FUNCTION_BLOCK FB_BagOpener
VAR_INPUT
  ams_net_id	: STRING;
END_VAR
VAR_OUTPUT
END_VAR
VAR
	adsread				: ADSREAD;
	adswrite			: ADSWRITE;
	status				: BagMachineStatus;
	iMethodTest			: BagMachineStatus;
	bagOpenStatus 		: BagMachineStatus;
  	error_code			: UINT;

	adsArr				: AdsArr;
	iState				: INT;
	iAds				: INT;
	ton_ms				: TON;
	iMachineStatus		: INT;//inArr[0]
	iBagStatus			: INT;//inArr[1]
	iBagDetectStatus	: INT;//inArr[2]
	iBagCmd				: INT;//outArr[1]
	iBagDetectCmd		: INT;//outArr[2]
	
	
	
END_VAR

	adsread(
			NETID:=ams_net_id , 
			PORT:=851 , 
			IDXGRP:=16#00004020 , 
			IDXOFFS:=100 , 
			LEN:= SIZEOF(adsArr.inArr), 
			DESTADDR:= ADR(adsArr.inArr), 
			READ:=, 
			TMOUT:=T#2S , 
			BUSY=> , 
			ERR=> , 
			ERRID=> );
	adswrite(
			NETID:=ams_net_id , 
			PORT:=851, 
			IDXGRP:=16#00004020, 
			IDXOFFS:=200, 
			LEN:=SIZEOF(adsArr.outArr) , 
			SRCADDR:=ADR(adsArr.outArr) , 
			WRITE:= , 
			TMOUT:=T#2S , 
			BUSY=> , 
			ERR=> , 
			ERRID=> );
ton_ms(PT:=T#2MS);			
CASE iAds OF 
	0:
		adsread.READ	:= FALSE;
		adswrite.WRITE	:= FALSE;	
		iAds	:=1;
	1:
		ton_ms.IN	:= TRUE;
		IF ton_ms.Q THEN
			ton_ms.IN	:= FALSE;
			iAds	:=2;
		END_IF
	2:
		adsread.READ	:= TRUE;
		adswrite.WRITE	:= TRUE;
		iAds	:=3;
	3:
		ton_ms.IN	:= TRUE;
		IF ton_ms.Q THEN
			ton_ms.IN	:= FALSE;
			iAds	:=0;
		END_IF	
END_CASE
//inputArr:
//		[0]:machine status;
//		[1]:bag status(3:BAG_READY,4:BAG_INSERTED,5:BAG_REMOVED,6:camera_ok,7:camera_ng);
//		[2]:bag detect status(0:idle,1:ok,2:ng);	
//outputArr:
//		[0]:line status;
//		[1]:bag cmd(1:insert_bag,2:bag_done_clamping,3:camera_trigger,4:camera_reset);
//	    [2]:bag detect cmd(0:idle,1:trigger,2:reset);
iMachineStatus		:= WORD_TO_INT(adsArr.inArr[0]);
iBagStatus 			:= WORD_TO_INT(adsArr.inArr[1]);
iBagDetectStatus	:= WORD_TO_INT(adsArr.inArr[2]);
adsArr.outArr[1]	:= INT_TO_WORD(iBagCmd);
adsArr.outArr[2]	:= INT_TO_WORD(iBagDetectCmd);

CASE iMachineStatus OF
	0:
		status	:= BagMachineStatus.OFF;
	1:
		status	:= BagMachineStatus.READY;
	2:
		status	:= BagMachineStatus.BUSY;
	3:
		status	:= BagMachineStatus.ERROR;
END_CASE
CASE iMethodTest OF
	BagMachineStatus.OFF:
		iState	:= BagMachineStatus.OFF;
	BagMachineStatus.BAG_INSERTED:
		IF GVL.fb_bagOpener.insert_bag() THEN
			iMethodTest	:=0;
		END_IF		
	BagMachineStatus.BAG_REMOVED:
		IF GVL.fb_bagOpener.bag_done_clamping() THEN
			iMethodTest	:=0;
		END_IF	
	BagMachineStatus.GET_RESULT_FROM_CAMERA:
		IF GVL.fb_bagOpener.getResultFromCamera() THEN
			iMethodTest	:=0;
		END_IF
	BagMachineStatus.RESET_CAMERA:
		IF GVL.fb_bagOpener.resetCamera() THEN
			iMethodTest	:=0;
		END_IF	
END_CASE
IF bag_ready THEN
	;
END_IF

{attribute 'TcRpcEnable'}
METHOD PUBLIC bag_done_clamping : BOOL
VAR_INPUT
END_VAR
bag_done_clamping	:= FALSE;
iBagCmd	:= BagCmd.REMOVE_ENABLE;
IF bag_removed OR bag_ready THEN//avoid not catch signal of removed
	bag_done_clamping	:= TRUE;
	iBagCmd	:= BagCmd.OFF;
END_IF
END_METHOD

PROPERTY bag_inserted : BOOL
GET
bag_inserted	:= (WORD_TO_INT(adsArr.inArr[1])	= BagMachineStatus.BAG_INSERTED);
END_GET
END_PROPERTY

PROPERTY bag_ready : BOOL
GET
bag_ready	:= (WORD_TO_INT(adsArr.inArr[1])	= BagMachineStatus.BAG_READY);
END_GET
END_PROPERTY

PROPERTY bag_removed : BOOL
GET
bag_removed	:= (WORD_TO_INT(adsArr.inArr[1])	= BagMachineStatus.BAG_REMOVED);
END_GET
END_PROPERTY

{attribute 'TcRpcEnable'}
METHOD PUBLIC getResultFromCamera : BOOL
VAR_INPUT

END_VAR
getResultFromCamera	:= FALSE;
CASE iState OF
	BagMachineStatus.OFF:
		IF iBagDetectStatus = BagMachineStatus.OFF THEN
			iState	:= BagMachineStatus.GET_RESULT_FROM_CAMERA;
		END_IF
	BagMachineStatus.GET_RESULT_FROM_CAMERA:
		iBagDetectCmd	:= 	BagCmd.GET_RESULT_FROM_CAMERA;
		IF iBagDetectStatus <> BagMachineStatus.OFF THEN
			getResultFromCamera	:= TRUE;
			iState	:= BagMachineStatus.OFF;
			iBagDetectCmd	:= 	BagCmd.OFF;
		END_IF	
	
END_CASE
END_METHOD

{attribute 'TcRpcEnable'}
METHOD PUBLIC insert_bag : BOOL
VAR_INPUT

END_VAR
insert_bag	:= FALSE;
CASE iState OF
	BagMachineStatus.OFF:
		iState	:= BagMachineStatus.BAG_READY;
	BagMachineStatus.BAG_READY:
		IF bag_ready THEN			
			iState	:= BagMachineStatus.BAG_INSERTED;
		END_IF		
	BagMachineStatus.BAG_INSERTED:
		iBagCmd	:= 	BagCmd.INSERT_ENABLE;
		IF bag_inserted THEN
			insert_bag	:= TRUE;
			iState	:= BagMachineStatus.OFF;
			iBagCmd	:= 	BagCmd.OFF;
		END_IF	
END_CASE
END_METHOD

METHOD M_Init : BOOL
VAR_INPUT
END_VAR
M_Init	:= FALSE;
iState	:= BagMachineStatus.OFF;
iBagDetectCmd	:= BagCmd.OFF;
iBagCmd	:= 	BagCmd.OFF;
M_Init	:= TRUE;
END_METHOD

{attribute 'TcRpcEnable'}
METHOD PUBLIC resetCamera : BOOL
VAR_INPUT

END_VAR
resetCamera	:= FALSE;
iBagDetectCmd	:= 	BagCmd.RESET_CAMERA;
IF iBagDetectStatus = BagMachineStatus.OFF THEN
	resetCamera	:= TRUE;
	iBagDetectCmd	:= 	BagCmd.OFF;
END_IF
END_METHOD

END_FUNCTION_BLOCK

(* stored: Version 1.1.0.1, ProductVersion 3.1.4024.12
   POU FB_BagOpener: Id {d990ddd1-9606-4745-b80b-134d02663290}, SpecialFunc None
   Method bag_done_clamping: Id {106afa9e-1515-436b-93db-b6ae6b065e5a}
   Property bag_inserted: Id {5d05c0dc-651b-47e9-9738-a91b3f9d748c}
   Get Get: Id {555689cb-662e-416b-955b-dd411e528cee}
   Property bag_ready: Id {997ca967-3d37-4a66-b58f-b695ba6a31b6}
   Get Get: Id {b4c37c5a-b78e-4308-ae60-eb17b4b6f6ab}
   Property bag_removed: Id {ac688585-3c93-428b-aa37-7290a5716161}
   Get Get: Id {398bd56f-f747-4f00-8c7a-3a6dc6d977b0}
   Method getResultFromCamera: Id {e17a1061-a312-4c90-ae11-f2c84b35ac55}
   Method insert_bag: Id {025d8fde-bab8-4359-812a-e6e638b46921}
   Method M_Init: Id {ab5f3fbb-59b8-4828-aeda-825e8bbd1b52}
   Method resetCamera: Id {ceb98418-f13a-4ed3-bbb0-590c0cc0059d} *)
